// TIA Portal V20 export
FUNCTION_BLOCK "Fx_Mixed"   // FB3, LAD
{ S7_Optimized_Access := 'TRUE' }
// stored: MemoryReserve 100, SetENOAutomatically false
   VAR_INPUT
      "a" : Int;
      "b" : Bool;
   END_VAR
   VAR_OUTPUT
      q : Int;
      r : Bool;
      s : Bool;
   END_VAR
BEGIN

REGION Network 1 (SCL)
   #q := #a * 2;
END_REGION

NETWORK
TITLE = 
      A     #"b";
      AN    #r;
      =     #s;
END_FUNCTION_BLOCK
